ABB RobotStudio station: MQP1.rsstn

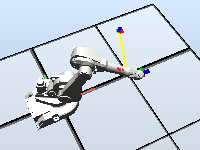
Station MQP1 (saved by RobotStudio 6.8.8148.134)
Controller System1
  mechanical unit ROB_1: IRB1600_6_120__02, 6 joints, base frame (0, 0, 0) mm
Layout (positions relative to the parent item):
  - IRB1600_6_120__02 [mechanism, from Robots\IRB1600_6_120_G_02.rslib] at (0, 0, 0) mm; joint values [-0.544, 0.5063, -0.1704, 2.0698, 0.6303, -2.1643] (rad or m)
Targets, tools, work objects and paths stored in the station, written as RAPID:
! task (no controller)
MODULE Module1
  CONST robtarget Target_20:=[[1000,0,0],[1,0,0,0],[0,0,0,0],[9E+09,9E+09,9E+09,9E+09,9E+09,9E+09]];
  CONST robtarget Target_30:=[[1000,0,0],[0.965925826,0.258819045,0,0],[0,0,0,0],[9E+09,9E+09,9E+09,9E+09,9E+09,9E+09]];
  CONST robtarget Target_40:=[[787.616,-60.118,993.149],[1,0,0,0],[0,0,0,0],[9E+09,9E+09,9E+09,9E+09,9E+09,9E+09]];
  PROC Path_10()
    MoveL Target_20,v1000,z100,tool0\WObj:=wobj0;
    MoveL Target_30,v1000,z100,tool0\WObj:=wobj0;
    MoveL Target_40,v1000,z100,tool0\WObj:=wobj0;
    MoveL Target_40,v1000,z100,tool0\WObj:=wobj0;
  ENDPROC
ENDMODULE

! task T_ROB1
MODULE Module1
  PROC Path_10()
  ENDPROC
ENDMODULE

